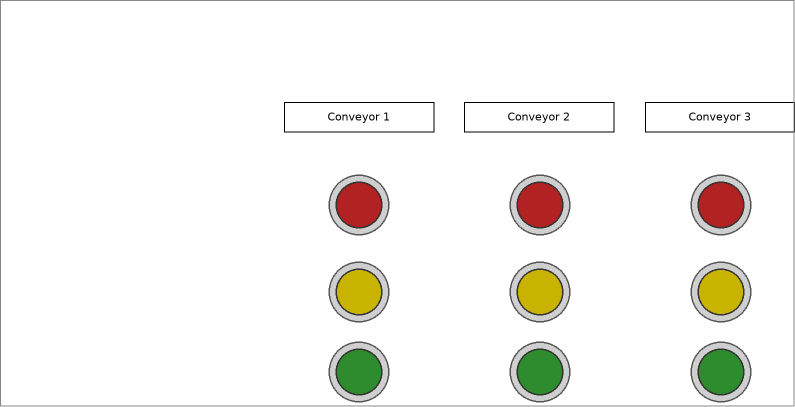
VISUALIZATION Visualization  // 795x407
    Lamp1 (324,170 70x70), variable: MAIN.conv1.red_light_on, style: Lamp-Lamp1-Red
    Lamp1 (324,257 70x70), variable: MAIN.conv1.yellow_light_on, style: Lamp-Lamp1-Yellow
    Lamp1 (324,337 70x70), variable: MAIN.conv1.green_light_on, style: Lamp-Lamp1-Green
    Lamp1 (505,170 70x70), variable: MAIN.conv2.red_light_on, style: Lamp-Lamp1-Red
    Lamp1 (505,257 70x70), variable: MAIN.conv2.yellow_light_on, style: Lamp-Lamp1-Yellow
    Lamp1 (505,337 70x70), variable: MAIN.conv2.green_light_on, style: Lamp-Lamp1-Green
    Lamp1 (686,170 70x70), variable: MAIN.conv3.red_light_on, style: Lamp-Lamp1-Red
    Lamp1 (686,257 70x70), variable: MAIN.conv3.yellow_light_on, style: Lamp-Lamp1-Yellow
    Lamp1 (686,337 70x70), variable: MAIN.conv3.green_light_on, style: Lamp-Lamp1-Green
    Rectangle (284,102 150x30), "Conveyor 1"
    Rectangle (464,102 150x30), "Conveyor 2"
    Rectangle (645,102 150x30), "Conveyor 3"
END_VISUALIZATION

(* stored: Version 1.1.0.1
   Visu Visualization: Id {475ef12b-6d56-44c1-8a7a-4a00b4733e70} *)
